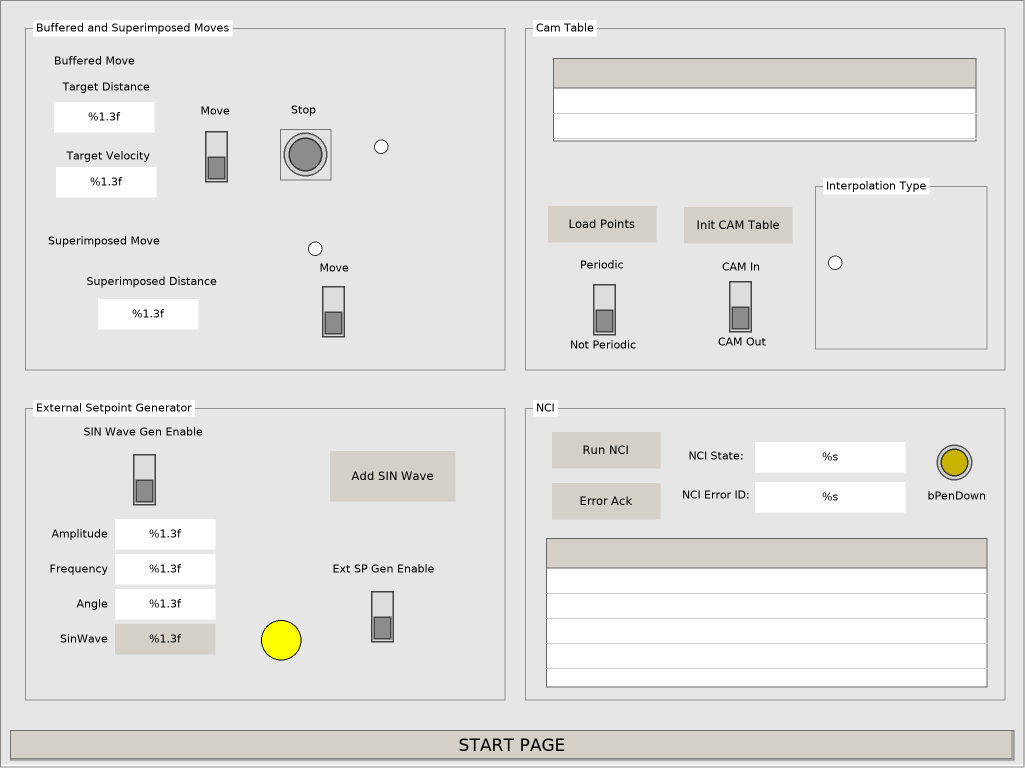
VISUALIZATION MotionProfiles  // 1025x768
    Rectangle (1,-4 1024x768)
    Button (10,730 1004x30), "START PAGE"
        OnMouseClick: change screen: HmiStartPage
    GroupBox (25,20 480x350), "Buffered and Superimposed Moves"
        Ellipse (236,600 40x40), colour toggle: Ext_SP_Gen.bAddSin
            toggle Ext_SP_Gen.bAddSin
        Label (12,30 115x22), "Buffered Move"
        Rectangle (29,82 100x30), "%1.3f", text variable: Axis3.lrMstrTarg2
            OnMouseDown: write the text variable via VisuDialogs.Numpad
        Rectangle (31,147 100x30), "%1.3f", text variable: Axis3.lrMstrVelo2
            OnMouseDown: write the text variable via VisuDialogs.Numpad
        Rectangle (30,56 98x22), "Target Distance"
        Rectangle (30,125 98x22), "Target Velocity"
        DipSwitch (166,108 51x57), variable: Axis3.bMvMstr2, behaviour: TOGGLE, style: Switch-DipSwitch-Gray
        RadioButton (347,95 96x63), variable: Axis3.iMstrMvMode2
            Areas[0]: Text=Absolute
            Areas[1]: Text=Relative
        PushSwitch (255,106 51x57), variable: Axis3.bStop, behaviour: TOGGLE, style: Switch-PushSwitch-Gray
        Label (12,210 134x22), "Superimposed Move"
        Label (159,80 63x22), "Move"
        Label (247,79 63x22), "Stop"
        Rectangle (73,279 100x30), "%1.3f", text variable: Axis3.lrMstrTarg3
            OnMouseDown: write the text variable via VisuDialogs.Numpad
        Rectangle (53,251 142x21), "Superimposed Distance"
        DipSwitch (283,263 51x57), variable: Axis3.bMvMstr2, behaviour: TOGGLE, style: Switch-DipSwitch-Gray
        Label (278,237 63x22), "Move"
    GroupBox (25,400 480x300), "External Setpoint Generator"
        DipSwitch (94,51 51x57), variable: Ext_SP_Gen.bSinGen, behaviour: TOGGLE, style: Switch-DipSwitch-Gray
        Label (45,21 147x22), "SIN Wave Gen Enable"
        DipSwitch (332,188 51x57), variable: Ext_SP_Gen.bMstrExtSP, behaviour: TOGGLE, style: Switch-DipSwitch-Gray
        Label (285,154 147x30), "Ext SP Gen Enable"
        Rectangle (11,158 75x22), "Frequency"
        Rectangle (305,51 125x50), "Add SIN Wave", colour toggle: Ext_SP_Gen.bAddSin
            toggle Ext_SP_Gen.bAddSin p2164770859=TRUE
    GroupBox (525,400 480x300), "NCI"
        Table (21,138 441x149), data array: NCI.aGCodeLines
            p3854506369: NCI.aGCodeLines[INDEX]
            p2232123230: Last 5 executed Gcode blocks
        Label (150,41 82x30), "NCI State:"
        Lamp1 (409,41 41x43), variable: NCI.bPenDown, style: Lamp-Lamp1-Yellow
        Rectangle (230,42 150x30), "%s", text variable: NCI.nNCI_State
        Label (150,80 82x30), "NCI Error ID:"
        Rectangle (230,82 150x30), "%s", text variable: NCI.nNciErrId
        Rectangle (27,32 108x36), "Run NCI", colour toggle: bRevSeqStart
            tap NCI.bRunNCI
        Rectangle (27,83 108x36), "Error Ack", colour toggle: bRevSeqStart
            tap NCI.bErrorAck
        Label (386,80 92x32), "bPenDown"
    GroupBox (525,20 480x350), "Cam Table"
        Rectangle (23,186 108x36), "Load Points", colour toggle: bRevSeqStart
            tap CamTable.bLoadPoints
        Rectangle (159,187 108x36), "Init CAM Table", colour toggle: bRevSeqStart
            tap CamTable.bCamInit
        DipSwitch (190,258 51x57), variable: CamTable.bCamIn, behaviour: TOGGLE, style: Switch-DipSwitch-Gray
        DipSwitch (54,261 51x57), variable: CamTable.bPeriodic, input disabled if: CamTable.bCamIn, behaviour: TOGGLE, style: Switch-DipSwitch-Gray
        Rectangle (168,311 98x22), "CAM Out"
        Rectangle (167,236 98x22), "CAM In"
        Rectangle (29,314 98x22), "Not Periodic"
        Rectangle (28,234 98x22), "Periodic"
        Table (28,38 423x83), data array: CamTable.arCamTable
            p3854506369: CamTable.arCamTable[0,INDEX]
            p1892666644: CamTable.arCamTable[1,INDEX]
            p338671338: CamTable.arCamTable[2,INDEX]
            p2170511999: CamTable.arCamTable[3,INDEX]
            p3723444502: CamTable.arCamTable[4,INDEX]
            p1218418051: CamTable.arCamTable[5,INDEX]
            p746581629: CamMotnFns.CamMotnFnPts[INDEX].SlavePos
            p3104783080: CamMotnFns.CamMotnFnPts[INDEX].SlaveVelo
            p2501879983: CamMotnFns.CamMotnFnPts[INDEX].SlaveAcc
            p7306298: CamMotnFns.CamMotnFnPts[INDEX].SlaveJerk
            p1137915858: CamTable.iSelY
            p1420305297: CamTable.iSelX
        GroupBox (290,158 172x171), "Interpolation Type"
            RadioButton (-509,19 137x103), variable: CamTable.iInterpType, input disabled if: CamTable.bCamIn
                Areas[0]: Text=Linear
                Areas[1]: Text=Spline
                Areas[2]: Text=Sliding Spline
        RadioButton (301,184 150x117), variable: CamTable.iInterpType, input disabled if: CamTable.bCamIn
            Areas[0]: Text=Linear
            Areas[1]: Text=Spline
            Areas[2]: Text=Sliding Spline
    Rectangle (115,624 100x30), "%1.3f", text variable: Ext_SP_Gen.lrSinWave
    Rectangle (115,589 100x30), "%1.3f", text variable: Ext_SP_Gen.rDeg
        OnMouseDown: write the text variable via VisuDialogs.Numpad
    Rectangle (58,593 53x22), "Angle"
    Rectangle (37,628 74x22), "SinWave"
    Rectangle (115,519 100x30), "%1.3f", text variable: Ext_SP_Gen.rSinAmp
        OnMouseDown: write the text variable via VisuDialogs.Numpad
    Rectangle (38,523 73x22), "Amplitude"
    Rectangle (115,554 100x30), "%1.3f", text variable: Ext_SP_Gen.rDegStep
        OnMouseDown: write the text variable via VisuDialogs.Numpad
END_VISUALIZATION

(* stored: Version 1.1.0.1
   Visu MotionProfiles: Id {0700ea4f-fdc5-4aac-a4ff-c4ee835689d8} *)
